{attribute 'linkalways'} 
{attribute 'no_explicit_call' := 'This FB is a CLASS and must be accessed using methods or properties'}
{attribute 'enable_dynamic_creation'}
FUNCTION_BLOCK Node_F_VN_MaxElementElementwise_ULINT EXTENDS VisionNode
VAR
    ipContainer : _ITcVnContainer;
    nMax : _ULINT(0);
    hrPrev : _HRESULT(S_OK);
    hresult : _HRESULT(S_OK);
END_VAR

METHOD PUBLIC  Clone : I_Node
VAR
	pNode : POINTER TO Node_F_VN_MaxElementElementwise_ULINT;
END_VAR
pNode := __NEW(Node_F_VN_MaxElementElementwise_ULINT);
Clone := pNode^;
END_METHOD

METHOD FB_init : BOOL
VAR_INPUT
	bInitRetains : BOOL; // if TRUE, the retain variables are initialized (warm start / cold start)
	bInCopyCode : BOOL;  // if TRUE, the instance afterwards gets moved into the copy code (online change)
END_VAR
AddInput('ipContainer', ipContainer);
AddInput('hrPrev', hrPrev);
AddOutput('ipContainer', ipContainer);
AddOutput('nMax', nMax);
AddOutput('hresult',hresult);
END_METHOD

METHOD PROTECTED OnExecute
hresult.Value := F_VN_MaxElementElementwise_ULINT(
    ipContainer := ipContainer.Value,
    nMax := nMax.Value,
    hrPrev:= hrPrev.Value);
END_METHOD

METHOD PUBLIC PreExecutionCheck
VAR_INPUT
	Check : I_PreExecutionChecks;
END_VAR
Check.IsTrue(ipContainer.IsValid, 'ipContainer must be a valid container');
Check.IsTrue(ipContainer.IsType(TC_GLOBAL_CONST_LIST.ContainerType_Vector_ULINT), 'ipContainer contains incorrect type');
END_METHOD

END_FUNCTION_BLOCK

(* stored: Version 1.1.0.1, ProductVersion 3.1.4026.13
   POU Node_F_VN_MaxElementElementwise_ULINT: Id {78a8fbe3-98fb-48b5-9231-a0494bfa8fdc}, SpecialFunc None
   Folder Constructor: Id {fc0e2590-3bc5-49a0-b7d9-6b1ff7bb6ca8}
   Method Clone: Id {04199cc4-bd47-4ad1-86d2-ea551f92102d}
   Method FB_init: Id {d25bdf1d-468e-43f0-8e05-113d35014aec}
   Method OnExecute: Id {cce3b198-d894-4137-9ddc-70ee835f4c92}
   Method PreExecutionCheck: Id {17a0be01-e5ca-428b-bf60-e1b9cfbb9922} *)
